(* PLC project ArrayDimProject *)

PROGRAM Main
  VAR
    BigArr : ARRAY[0..100000000] OF REAL;
    SmallArr : ARRAY[1..8] OF INT;
  END_VAR


END_PROGRAM

CONFIGURATION Config
  RESOURCE Res ON PLC
  END_RESOURCE
END_CONFIGURATION
